INTERFACE ITFGesimuleerdAI

PROPERTY SensorWaarde : int
GET
END_GET
SET
END_SET
END_PROPERTY

END_INTERFACE

(* stored: Version 1.1.0.1
   Itf ITFGesimuleerdAI: Id {37c3b61f-23f6-47a0-bbb9-132e2ec031f5}
   Property SensorWaarde: Id {355f3bf6-447b-4733-9e51-49350e9b7c8f}
   Get Get: Id {d19fda89-9ee2-4f7e-8e7b-f5f5f758b1c0}
   Set Set: Id {4cdb3660-85d4-426f-987f-afd42a6688ec} *)
